MOVL C01141 V=30.0 PL=1
CALL JOB:EXTRUDE
MOVL C01142 V=30.0 PL=1
CALL JOB:EXTRUDE
MOVL C01143 V=30.0 PL=1
MOVL C01144 V=130.0 PL=1
MOVL C01145 V=130.0 PL=1
CALL JOB:EXTRUDE
MOVL C01146 V=20.0 PL=1
MOVL C01147 V=130.0 PL=1
MOVL C01148 V=130.0 PL=1
CALL JOB:EXTRUDE
MOVL C01149 V=60.0 PL=1
CALL JOB:EXTRUDE
MOVL C01150 V=60.0 PL=1
CALL JOB:EXTRUDE
MOVL C01151 V=60.0 PL=1
CALL JOB:EXTRUDE
MOVL C01152 V=60.0 PL=1
MOVL C01153 V=130.0 PL=1
CALL JOB:EXTRUDE
MOVL C01154 V=30.0 PL=1
CALL JOB:EXTRUDE
MOVL C01155 V=30.0 PL=1
CALL JOB:EXTRUDE
MOVL C01156 V=30.0 PL=1
CALL JOB:EXTRUDE
MOVL C01157 V=30.0 PL=1
CALL JOB:EXTRUDE
MOVL C01158 V=30.0 PL=1
CALL JOB:EXTRUDE
MOVL C01159 V=30.0 PL=1
CALL JOB:EXTRUDE
MOVL C01160 V=30.0 PL=1
END
